Staubli VAL3: iSample.pgx

public program iSample(num& nNum[] (dimensions=1))
begin
  nNum=dioGet(iSampleStatus)
end
